PROGRAM MAIN
VAR
	
	firstCycle	: BOOL := TRUE;
	fb_Time : FB_LocalSystemTime;
	Temp_str : STRING;
   	
	
	str_state	: STRING;
	application	: FB_Application;
	rtReset		: R_TRIG;
	rtInit		: R_TRIG;
	rtRun		: R_TRIG;
	rtSafety	: R_TRIG;
	
	ton_timeout			: TON;	
	eState				: E_SystemManager	:= E_SystemManager.START;
	eStateTemp			: E_SystemManager	:= E_SystemManager.START;
	iStateTemp			: INT;
	sStateTemp			: STRING;	
	
	
	auto_store_run		: BOOL;
	auto_store_sensor	: BOOL;
	rtStop_auto_store	: R_TRIG;
	bButton				: BOOL;
	ton_button			: TON;
	resetting			: BOOL;
	initializing		: BOOL;
	running				: BOOL;
	
	
	pMachine_status	: POINTER TO MachineStatus;
	pMachine_control_cmd	: POINTER TO MachineControlCommand;
	b_test: BOOL;
	event	: ST_EVENT;
	b_test1: BOOL;
END_VAR

//////////////////////////////////////////////////////////timeout//////////////////////////////////////////
iStateTemp	:= eStateTemp;
sStateTemp	:= INT_TO_STRING(iStateTemp);
ton_timeout();
IF eState<>E_SystemManager.START AND eState<>E_SystemManager.ERROR THEN
	IF eStateTemp=eState THEN
		ton_timeout.IN	:=TRUE;
	ELSE
		ton_timeout.IN	:=FALSE;
		eStateTemp	:= eState;	
	END_IF
ELSE
	ton_timeout.IN	:=FALSE;
END_IF
IF ton_timeout.Q THEN	
	ton_timeout.IN	:=FALSE;
	CASE eState OF		
		E_SystemManager.START:
			;	
		
	END_CASE
//	IF eStates<>E_WorkingStates.WAIT_NEW_TOTE AND eStates<>E_WorkingStates.WAIT THEN
//		eStates	:= E_WorkingStates.ERROR;
//	END_IF
	
END_IF


IF firstCycle THEN
	firstCycle := FALSE;
END_IF
pMachine_status	:= ADR(MAIN.application.tote_subsystem.status);
pMachine_control_cmd	:= ADR(MAIN.application.tote_subsystem.machine_control_cmd);
fb_Time(bEnable := TRUE);
Temp_str := Prepare_Date_Time(fb_Time.systemTime);
rtSafety(CLK:=application.safety.xError);
rtReset(CLK:=G_HMI.bReset OR GVL.fb_mcp.st_safety_door.button_reset OR pMachine_control_cmd^=MachineControlCommand.RESET);
rtInit(CLK:=G_HMI.bInit);
rtRun(CLK:=G_HMI.bRun);

IF rtSafety.Q THEN
	eState	:= E_SystemManager.ERROR_SAFETY;
END_IF
(******************************************************************************
State Machine
******************************************************************************)
//error while running than estate=error,if electrical error,trig xerror and estate=error
//reset: xError->false and reset devices
//wait 1s,
CASE eState OF
	E_SystemManager.START:
		;
	E_SystemManager.INITIALIZATION:
		;
	E_SystemManager.RESET:
		eState	:= E_SystemManager.RESET_SAFETY;
	E_SystemManager.RESET_SAFETY:
		ton_timeout.PT:= T#2S;
		IF application.safety.M_reset() THEN
			IF application.safety.xError THEN
				eState	:= E_SystemManager.ERROR_SAFETY;
			ELSE
				eState	:= E_SystemManager.RESET_FB_LOADING;
			END_IF
		END_IF
	E_SystemManager.RESET_FB_LOADING:
		IF GVL.fb_loading.M_reset() THEN
			IF GVL.fb_loading.xError THEN
				eState	:= E_SystemManager.ERROR;
			ELSE
				eState	:= E_SystemManager.RESET_FB_BUFFER;
			END_IF
		END_IF
	E_SystemManager.RESET_FB_BUFFER:
		IF GVL.fb_buffer.M_reset() THEN
			IF GVL.fb_buffer.xError THEN
				eState	:= E_SystemManager.ERROR;
			ELSE
				eState	:= E_SystemManager.RESET_FB_WORKING;
			END_IF
		END_IF		
	E_SystemManager.RESET_FB_WORKING:
		IF GVL.fb_working.M_reset() THEN
			IF GVL.fb_working.xError THEN
				eState	:= E_SystemManager.ERROR;
			ELSE
				eState	:= E_SystemManager.READY;
			END_IF
		END_IF		
		
	E_SystemManager.INIT_SAFETY:
		IF application.safety.M_reset() THEN
			IF application.safety.xError THEN
				eState	:= E_SystemManager.ERROR_SAFETY;
			ELSE
				eState	:= E_SystemManager.INIT_FB_LOADING;
			END_IF
		END_IF
	E_SystemManager.INIT_FB_LOADING:
		IF GVL.fb_loading.M_init() THEN
			IF GVL.fb_loading.xError THEN
				eState	:= E_SystemManager.ERROR;
			ELSE
				eState	:= E_SystemManager.INIT_FB_BUFFER;
			END_IF
		END_IF
	E_SystemManager.INIT_FB_BUFFER:
		IF GVL.fb_buffer.M_init() THEN
			IF GVL.fb_buffer.xError THEN
				eState	:= E_SystemManager.ERROR;
			ELSE
				eState	:= E_SystemManager.INIT_FB_WORKING;
			END_IF
		END_IF		
	E_SystemManager.INIT_FB_WORKING:
		IF GVL.fb_working.M_init() THEN
			IF GVL.fb_working.xError THEN
				eState	:= E_SystemManager.ERROR;
			ELSE
				eState	:= E_SystemManager.RESET_SAFETY;
			END_IF
		END_IF				
		
	E_SystemManager.READY:
		eState	:= E_SystemManager.READY_TO_JOB;//todo add condition to jump to ready_to_job
	E_SystemManager.READY_TO_JOB://todo add condition to jump to ready
		pMachine_status^	:= MachineStatus.READY;
		IF G_HMI.bRun OR pMachine_control_cmd^=MachineControlCommand.START THEN
			pMachine_control_cmd^	:= MachineControlCommand.DO_NOTHING;
			GVL.bRunning	:= TRUE;
			eState	:= E_SystemManager.RUN_START;
		END_IF
		IF G_HMI.bAging_test THEN
			eState	:= E_SystemManager.AGAING_TEST;
		END_IF
	E_SystemManager.BUSY:
		;
	E_SystemManager.RUN_START:
		GVL.fb_buffer.M_runStart();
		GVL.fb_loading.M_runStart();
		GVL.fb_working.M_runStart();
		eState	:= E_SystemManager.IN_PROGRESS;
		GVL.bRunning	:= TRUE;
	E_SystemManager.IN_PROGRESS:
		pMachine_status^ := MachineStatus.RUNNING;
		GVL.fb_buffer.M_run();
		GVL.fb_loading.M_run();
		IF pMachine_control_cmd^=MachineControlCommand.STOP OR G_HMI.bStop THEN
			GVL.bRunning	:= FALSE;
			GVL.bAck_stop	:= TRUE;
			pMachine_control_cmd^	:= MachineControlCommand.DO_NOTHING;
		END_IF
		IF GVL.bAck_stop THEN
			IF pMachine_control_cmd^=MachineControlCommand.START OR G_HMI.bRun THEN
				GVL.bRunning	:= TRUE;
				GVL.bAck_stop	:= FALSE;
				pMachine_control_cmd^	:= MachineControlCommand.DO_NOTHING;
			END_IF
		END_IF		
		IF M_checkError() THEN
			GVL.fb_buffer.M_safetyEvent();
			GVL.fb_loading.M_safetyEvent();
			GVL.fb_working.M_safetyEvent();
			eState	:= E_SystemManager.ERROR;
		END_IF
	
	E_SystemManager.ERROR:
		pMachine_status^	:= MachineStatus.ERROR;
		IF rtReset.Q THEN
			Event_clear();
			pMachine_status^	:= MachineStatus.RESETTING;
			pMachine_control_cmd^	:= MachineControlCommand.DO_NOTHING;
			eState	:= E_SystemManager.RESET_SAFETY;
		END_IF
		IF rtInit.Q THEN
			pMachine_status^	:= MachineStatus.INITIALIZING;
			Event_clear();
			eState	:= E_SystemManager.INIT_SAFETY;					
		END_IF		
	E_SystemManager.ERROR_SAFETY:
		GVL.fb_buffer.M_safetyEvent();
		GVL.fb_loading.M_safetyEvent();
		GVL.fb_working.M_safetyEvent();
		eState	:= E_SystemManager.ERROR;
	E_SystemManager.REJECT:
		; 
	E_SystemManager.ON_POWER://	============================================================================== 
		;							//Check if components and tools ready to state REJECT,else to State ERROR								//check if reject is done then go to ready, else go to error state	
	E_SystemManager.AGAING_TEST:
		GVL.fb_buffer.M_agingTest();
		GVL.fb_loading.M_agingTest();
		GVL.fb_working.M_agingTest();
END_CASE

IF eState<>E_SystemManager.IN_PROGRESS THEN
	GVL.bAck_stop	:= FALSE;
	GVL.bRunning	:= FALSE;
END_IF
//////////////////////////////////////////////////////////mapping//////////////////////////////////////////
GVL.fb_working(	pre_tote_status:= GVL.fb_loading.current_tote_status);
GVL.fb_loading(	pre_tote_status:=GVL.fb_buffer.fb_rollers[3].current_tote_status,
				next_tote_status:=GVL.fb_working.current_tote_status);
GVL.fb_buffer();
GVL.fb_mcp();
M_convert_estate_string(eState:=eState,str_state=>str_state);

application();



auto_store_simulation();

IF b_test THEN
	event.sTime	:= MAIN.Temp_str;
	event.sComponent_name	:='test';
	event.sEvent_MSG	:='alarm test';
	Event_add(event);
	b_test	:= FALSE;
END_IF
IF b_test1 THEN
	Event_clear();
END_IF

ACTION auto_store_simulation:
G_IO.arDO[0].Ch[13]	:= auto_store_run;
auto_store_sensor	:= G_IO.arDI[0].Ch[13];
bButton				:= G_IO.arDI[0].Ch[14];
ton_button(IN:=bButton,PT:=T#2S);
rtStop_auto_store(CLK:=auto_store_sensor);
IF ton_button.Q THEN
	auto_store_run	:= TRUE;
END_IF
IF rtStop_auto_store.Q THEN
	auto_store_run	:= FALSE;
END_IF
IF application.safety.xError THEN
	auto_store_run	:= FALSE;
END_IF
END_ACTION

METHOD M_checkError : BOOL
VAR_INPUT
END_VAR



M_checkError	:= GVL.fb_buffer.xError OR GVL.fb_loading.xError OR GVL.fb_working.xError;
END_METHOD

METHOD M_convert_estate_string : BOOL
VAR_INPUT
	eState	:E_SystemManager;
END_VAR
VAR_OUTPUT
	str_state	: STRING;
END_VAR
CASE eState OF
	E_SystemManager.START:
		str_state	:= 'START';
	E_SystemManager.INITIALIZATION:
		str_state	:= 'INITIALIZATION';
	E_SystemManager.RESET:
		str_state	:= 'RESET';
	E_SystemManager.RESET_SAFETY:
		str_state	:= 'RESET_SAFETY';
	E_SystemManager.RESET_FB_LOADING:
		str_state	:= 'RESET_FB_LOADING';
	E_SystemManager.RESET_FB_BUFFER:
		str_state	:= 'RESET_FB_BUFFER';	
	E_SystemManager.RESET_FB_WORKING:
		str_state	:= 'RESET_FB_WORKING';
	E_SystemManager.INIT_SAFETY:
		str_state	:= 'INIT_SAFETY';
	E_SystemManager.INIT_FB_LOADING:
		str_state	:= 'INIT_FB_LOADING';
	E_SystemManager.INIT_FB_BUFFER:
		str_state	:= 'INIT_FB_BUFFER';
	E_SystemManager.INIT_FB_WORKING:			
		str_state	:= 'INIT_FB_WORKING';		
	E_SystemManager.READY:
		str_state	:= 'READY';
	E_SystemManager.READY_TO_JOB:
		str_state	:= 'READY_TO_JOB';
	E_SystemManager.BUSY:
		str_state	:= 'BUSY';
	E_SystemManager.RUN_START:
		str_state	:= 'RUN_START';
	E_SystemManager.IN_PROGRESS:
		str_state	:= 'IN_PROGRESS';
	E_SystemManager.ERROR:
		str_state	:= 'ERROR';
	E_SystemManager.ERROR_SAFETY:
		str_state	:= 'ERROR_SAFETY';
	E_SystemManager.REJECT:
		str_state	:= 'REJECT';
	E_SystemManager.ON_POWER://	============================================================================== 
		str_state	:= 'ON_POWER';
	E_SystemManager.AGAING_TEST:
		str_state	:= 'AGAING_TEST';
END_CASE
END_METHOD

END_PROGRAM

(* stored: Version 1.1.0.1, ProductVersion 3.1.4024.12
   POU MAIN: Id {ec74ff4b-2541-4a74-9976-19374303195a}, SpecialFunc None
   Action auto_store_simulation: Id {5e7c4530-8faf-4286-a590-f7a53f75013f}
   Method M_checkError: Id {2a7b0736-01e7-4929-a7b3-7cc5bb04f63e}
   Method M_convert_estate_string: Id {8c9fd5ea-f1d3-49b9-a404-1083d89866f2} *)
